FUNCTION_BLOCK EL3048
VAR
	_io : EL3xx8_Data;
	{attribute addProperty Name "WcState"}
	_wcState : WcStateInputToggle;
	{attribute addProperty Name "Info data"}
	_infoData : InfoDataAds;
END_VAR

PROPERTY IO : REFERENCE TO EL3xx8_Data
GET
IO REF= _io;
END_GET
END_PROPERTY

PROPERTY WcState : REFERENCE TO WcStateInputToggle
GET
WcState REF= _wcState;
END_GET
END_PROPERTY

END_FUNCTION_BLOCK

(* stored: Version 1.1.0.1, ProductVersion 3.1.4024.9
   POU EL3048: Id {07ab9aec-8b6b-0cea-2f55-67c2947d4027}, SpecialFunc None
   Property IO: Id {1e407642-d228-0aad-3747-0e54840908fb}
   Get Get: Id {2beeae3e-4305-039f-3822-48237f951689}
   Property WcState: Id {a88294ad-fbaf-059b-22b5-9cbf75cf693c}
   Get Get: Id {1b27425f-4857-05ac-12f8-69136fba9dde} *)
